FUNCTION_BLOCK FB_EZylinder
VAR_INPUT
	bGate : BOOL;
	bError : BOOL;
END_VAR
VAR_OUTPUT
	bR1 : BOOL;
	bR2 : BOOL;
END_VAR
VAR
END_VAR

bR1 := bGate;
bR2 := NOT bGate;

IF bError THEN
	bR1 := FALSE;
	bR2 := FALSE;
END_IF

END_FUNCTION_BLOCK

(* stored: Version 1.1.0.1, ProductVersion 3.1.4024.15
   POU FB_EZylinder: Id {829d8215-b376-445a-9de1-443716633f26}, SpecialFunc None *)
